{attribute 'GeneratedUsingTerminal: EL3483-0000-0016'}
{attribute addProperty BoxType "EL3483-0000-0016"}
{attribute addProperty Id "System_StateAT %I*BOOL1Grid_DirectionAT %I*BOOL1Frequency_Guard_WarningAT %I*BOOL1Frequency_Guard_ErrorAT %I*BOOL1Power_Quality_Guard_WarningAT %I*BOOL1Power_Quality_Guard_ErrorAT %I*BOOL1TxPDO_StateAT %I*BOOL1TxPDO_ToggleAT %I*BOOL1Power_Quality_FactorAT %I*REAL4"}
{attribute addProperty CRC "2906899385"}
{attribute addProperty Size "12"}
TYPE Total_Status_AD43C3B9 EXTENDS InputBase_8311D824 :
STRUCT
	{attribute addProperty Name "System_State"}
	System_State AT %I* : BOOL;
	{attribute addProperty Name "Grid_Direction"}
	Grid_Direction AT %I* : BOOL;
	{attribute addProperty Name "Frequency_Guard_Warning"}
	Frequency_Guard_Warning AT %I* : BOOL;
	{attribute addProperty Name "Frequency_Guard_Error"}
	Frequency_Guard_Error AT %I* : BOOL;
	{attribute addProperty Name "Power_Quality_Guard_Warning"}
	Power_Quality_Guard_Warning AT %I* : BOOL;
	{attribute addProperty Name "Power_Quality_Guard_Error"}
	Power_Quality_Guard_Error AT %I* : BOOL;
	{attribute addProperty Name "TxPDO_State"}
	TxPDO_State AT %I* : BOOL;
	{attribute addProperty Name "TxPDO_Toggle"}
	TxPDO_Toggle AT %I* : BOOL;
	{attribute addProperty Name "Power_Quality_Factor"}
	Power_Quality_Factor AT %I* : REAL;
END_STRUCT
END_TYPE

(* stored: Version 1.2.0.0, ProductVersion 3.1.4024.9
   DUT Total_Status_AD43C3B9: Id {01c6b65f-379c-42b8-85a9-22f923b28733} *)
